// TIA Portal V16 program export: 2 tag tables, 1 data types, 0 data blocks, 8 code blocks (in call order from the OBs), 7 instance data blocks

VAR_GLOBAL   // PLC tag table "Default tag table"
END_VAR

VAR_GLOBAL   // PLC tag table "Outputs"
   qIO_xSupplyConveyor1 AT %Q0.0 : Bool;
   qIO_xSupplyConveyor2 AT %Q0.1 : Bool;
   qIO_xS1Conveyor1 AT %Q0.2 : Bool;
   qIO_xS1Conveyor2 AT %Q0.3 : Bool;
   qIO_xS1Conveyor3 AT %Q0.4 : Bool;
   qIO_xS1PositionerClamp AT %Q0.5 : Bool;
   qIO_xS1PositionerRaise AT %Q0.6 : Bool;
   qIO_xS2Conveyor1 AT %Q0.7 : Bool;
   qIO_xS2Conveyor2 AT %Q1.0 : Bool;
   qIO_xS2Conveyor3 AT %Q1.1 : Bool;
   qIO_xS2PositionerClamp AT %Q1.2 : Bool;
   qIO_xS2PositionerRaise AT %Q1.3 : Bool;
   qIO_xS3Conveyor1 AT %Q1.4 : Bool;
   qIO_xS3Conveyor2 AT %Q1.5 : Bool;
   qIO_xS3Conveyor3 AT %Q1.6 : Bool;
   qIO_xS3PositionerClamp AT %Q1.7 : Bool;
   qIO_xS3PositionerRaise AT %Q2.0 : Bool;
   qIO_xS1ProcessLight AT %Q2.1 : Bool;
   qIO_iS1ProcessTimeLeft AT %QD10 : DInt;
   qIO_xS2ProcessLight AT %Q2.2 : Bool;
   qIO_iS2ProcessTimeLeft AT %QD14 : DInt;
   qIO_xS3ProcessLight AT %Q2.3 : Bool;
   qIO_iS3ProcessTimeLeft AT %QD18 : DInt;
   qIO_xSupplyGetMaterial AT %Q2.4 : Bool;
END_VAR

TYPE "UDT SupplyStation"
// stored: IsFailsafeCompliant false
   STRUCT
      Status : Struct
         xSpare : Bool;
      END_STRUCT;
      Command : Struct
         xSupplyDataRequest : Bool;
      END_STRUCT;
      Fault : Struct
         xSpare : Bool;
      END_STRUCT;
   END_STRUCT;
END_TYPE

ORGANIZATION_BLOCK "Main"   // OB1, LAD, ProgramCycle
TITLE = "Main Program Sweep (Cycle)"
{ S7_Optimized_Access := 'TRUE' }
VERSION : 0.1
// stored: AutoNumber true, IsIECCheckEnabled false, SetENOAutomatically false
   VAR_INPUT
      Initial_Call : Bool;   // Initial call of this OB
      Remanence : Bool;   // =True, if remanent data are available
   END_VAR
   VAR_TEMP   // added for the SCL form of the ladder/FBD networks
      _w1 : Bool;
   END_VAR
BEGIN

REGION Network 1
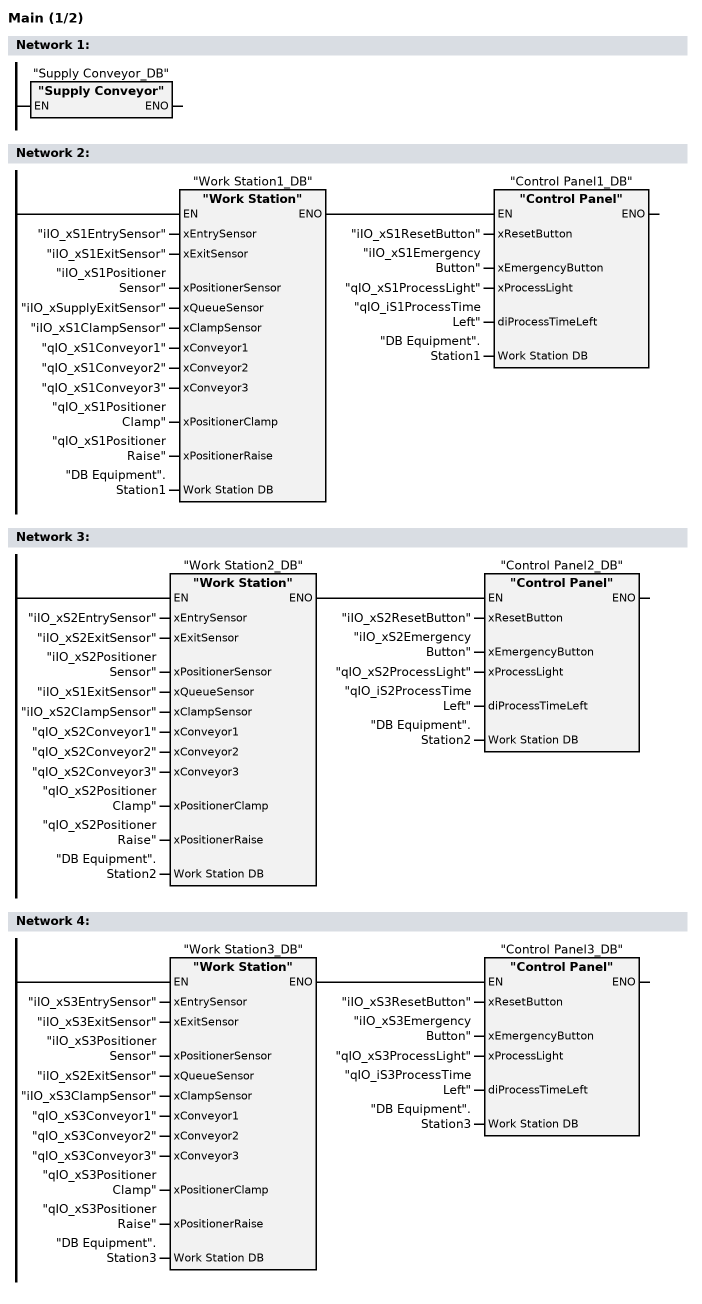
   RUNG wire#powerrail
      "Supply Conveyor_DB"()
   END_RUNG
   // the same network as SCL:
   "Supply Conveyor_DB"();   // "Supply Conveyor"
END_REGION

REGION Network 2
   RUNG wire#powerrail
      "Work Station1_DB"(xEntrySensor := "iIO_xS1EntrySensor", xExitSensor := "iIO_xS1ExitSensor", xPositionerSensor := "iIO_xS1PositionerSensor", xQueueSensor := "iIO_xSupplyExitSensor", xClampSensor := "iIO_xS1ClampSensor", xConveyor1 := "qIO_xS1Conveyor1", xConveyor2 := "qIO_xS1Conveyor2", xConveyor3 := "qIO_xS1Conveyor3", xPositionerClamp := "qIO_xS1PositionerClamp", xPositionerRaise := "qIO_xS1PositionerRaise", "Work Station DB" := "DB Equipment".Station1)
      "Control Panel1_DB"(xResetButton := "iIO_xS1ResetButton", xEmergencyButton := "iIO_xS1EmergencyButton", xProcessLight := "qIO_xS1ProcessLight", diProcessTimeLeft := "qIO_iS1ProcessTimeLeft", "Work Station DB" := "DB Equipment".Station1)
   END_RUNG
   // the same network as SCL:
   "Work Station1_DB"(xEntrySensor := "iIO_xS1EntrySensor",   // "Work Station"
                      xExitSensor := "iIO_xS1ExitSensor",
                      xPositionerSensor := "iIO_xS1PositionerSensor",
                      xQueueSensor := "iIO_xSupplyExitSensor",
                      xClampSensor := "iIO_xS1ClampSensor",
                      xConveyor1 := "qIO_xS1Conveyor1",
                      xConveyor2 := "qIO_xS1Conveyor2",
                      xConveyor3 := "qIO_xS1Conveyor3",
                      xPositionerClamp := "qIO_xS1PositionerClamp",
                      xPositionerRaise := "qIO_xS1PositionerRaise",
                      "Work Station DB" := "DB Equipment".Station1,
                      ENO => #_w1);
   IF #_w1 THEN
       "Control Panel1_DB"(xResetButton := "iIO_xS1ResetButton",   // "Control Panel"
                           xEmergencyButton := "iIO_xS1EmergencyButton",
                           xProcessLight := "qIO_xS1ProcessLight",
                           diProcessTimeLeft := "qIO_iS1ProcessTimeLeft",
                           "Work Station DB" := "DB Equipment".Station1);
   END_IF;
END_REGION

REGION Network 3
   RUNG wire#powerrail
      "Work Station2_DB"(xEntrySensor := "iIO_xS2EntrySensor", xExitSensor := "iIO_xS2ExitSensor", xPositionerSensor := "iIO_xS2PositionerSensor", xQueueSensor := "iIO_xS1ExitSensor", xClampSensor := "iIO_xS2ClampSensor", xConveyor1 := "qIO_xS2Conveyor1", xConveyor2 := "qIO_xS2Conveyor2", xConveyor3 := "qIO_xS2Conveyor3", xPositionerClamp := "qIO_xS2PositionerClamp", xPositionerRaise := "qIO_xS2PositionerRaise", "Work Station DB" := "DB Equipment".Station2)
      "Control Panel2_DB"(xResetButton := "iIO_xS2ResetButton", xEmergencyButton := "iIO_xS2EmergencyButton", xProcessLight := "qIO_xS2ProcessLight", diProcessTimeLeft := "qIO_iS2ProcessTimeLeft", "Work Station DB" := "DB Equipment".Station2)
   END_RUNG
   // the same network as SCL:
   "Work Station2_DB"(xEntrySensor := "iIO_xS2EntrySensor",   // "Work Station"
                      xExitSensor := "iIO_xS2ExitSensor",
                      xPositionerSensor := "iIO_xS2PositionerSensor",
                      xQueueSensor := "iIO_xS1ExitSensor",
                      xClampSensor := "iIO_xS2ClampSensor",
                      xConveyor1 := "qIO_xS2Conveyor1",
                      xConveyor2 := "qIO_xS2Conveyor2",
                      xConveyor3 := "qIO_xS2Conveyor3",
                      xPositionerClamp := "qIO_xS2PositionerClamp",
                      xPositionerRaise := "qIO_xS2PositionerRaise",
                      "Work Station DB" := "DB Equipment".Station2,
                      ENO => #_w1);
   IF #_w1 THEN
       "Control Panel2_DB"(xResetButton := "iIO_xS2ResetButton",   // "Control Panel"
                           xEmergencyButton := "iIO_xS2EmergencyButton",
                           xProcessLight := "qIO_xS2ProcessLight",
                           diProcessTimeLeft := "qIO_iS2ProcessTimeLeft",
                           "Work Station DB" := "DB Equipment".Station2);
   END_IF;
END_REGION

REGION Network 4
   RUNG wire#powerrail
      "Work Station3_DB"(xEntrySensor := "iIO_xS3EntrySensor", xExitSensor := "iIO_xS3ExitSensor", xPositionerSensor := "iIO_xS3PositionerSensor", xQueueSensor := "iIO_xS2ExitSensor", xClampSensor := "iIO_xS3ClampSensor", xConveyor1 := "qIO_xS3Conveyor1", xConveyor2 := "qIO_xS3Conveyor2", xConveyor3 := "qIO_xS3Conveyor3", xPositionerClamp := "qIO_xS3PositionerClamp", xPositionerRaise := "qIO_xS3PositionerRaise", "Work Station DB" := "DB Equipment".Station3)
      "Control Panel3_DB"(xResetButton := "iIO_xS3ResetButton", xEmergencyButton := "iIO_xS3EmergencyButton", xProcessLight := "qIO_xS3ProcessLight", diProcessTimeLeft := "qIO_iS3ProcessTimeLeft", "Work Station DB" := "DB Equipment".Station3)
   END_RUNG
   // the same network as SCL:
   "Work Station3_DB"(xEntrySensor := "iIO_xS3EntrySensor",   // "Work Station"
                      xExitSensor := "iIO_xS3ExitSensor",
                      xPositionerSensor := "iIO_xS3PositionerSensor",
                      xQueueSensor := "iIO_xS2ExitSensor",
                      xClampSensor := "iIO_xS3ClampSensor",
                      xConveyor1 := "qIO_xS3Conveyor1",
                      xConveyor2 := "qIO_xS3Conveyor2",
                      xConveyor3 := "qIO_xS3Conveyor3",
                      xPositionerClamp := "qIO_xS3PositionerClamp",
                      xPositionerRaise := "qIO_xS3PositionerRaise",
                      "Work Station DB" := "DB Equipment".Station3,
                      ENO => #_w1);
   IF #_w1 THEN
       "Control Panel3_DB"(xResetButton := "iIO_xS3ResetButton",   // "Control Panel"
                           xEmergencyButton := "iIO_xS3EmergencyButton",
                           xProcessLight := "qIO_xS3ProcessLight",
                           diProcessTimeLeft := "qIO_iS3ProcessTimeLeft",
                           "Work Station DB" := "DB Equipment".Station3);
   END_IF;
END_REGION

REGION Network 5
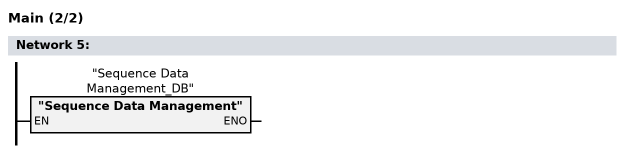
   RUNG wire#powerrail
      "Sequence Data Management_DB"()
   END_RUNG
   // the same network as SCL:
   "Sequence Data Management_DB"();   // "Sequence Data Management"
END_REGION
END_ORGANIZATION_BLOCK

FUNCTION_BLOCK "Work Station"   // FB1, LAD
{ S7_Optimized_Access := 'TRUE' }
VERSION : 0.1
// stored: AutoNumber true, IsIECCheckEnabled false, IsRetainMemResEnabled false, MemoryReserve 100, SetENOAutomatically false, UDAEnableTagReadback false
   VAR_INPUT
      xEntrySensor { ExternalAccessible := 'False'; ExternalVisible := 'False'; ExternalWritable := 'False'} : Bool;
      xExitSensor { ExternalAccessible := 'False'; ExternalVisible := 'False'; ExternalWritable := 'False'} : Bool;
      xPositionerSensor { ExternalAccessible := 'False'; ExternalVisible := 'False'; ExternalWritable := 'False'} : Bool;
      xQueueSensor { ExternalAccessible := 'False'; ExternalVisible := 'False'; ExternalWritable := 'False'} : Bool;
      xClampSensor { ExternalAccessible := 'False'; ExternalVisible := 'False'; ExternalWritable := 'False'} : Bool;
   END_VAR
   VAR_IN_OUT
      xConveyor1 { ExternalAccessible := 'False'; ExternalVisible := 'False'; ExternalWritable := 'False'} : Bool;
      xConveyor2 { ExternalAccessible := 'False'; ExternalVisible := 'False'; ExternalWritable := 'False'} : Bool;
      xConveyor3 { ExternalAccessible := 'False'; ExternalVisible := 'False'; ExternalWritable := 'False'} : Bool;
      xPositionerClamp : Bool;
      xPositionerRaise : Bool;
      "Work Station DB" : "UDT WorkStation";
   END_VAR
   VAR
      StationConveyorControl_Instance { S7_SetPoint := 'True'} : "StationConveyorControl";
      StationProcessControl_Instance { S7_SetPoint := 'True'} : "StationProcessControl";
   END_VAR
BEGIN

REGION Network 2
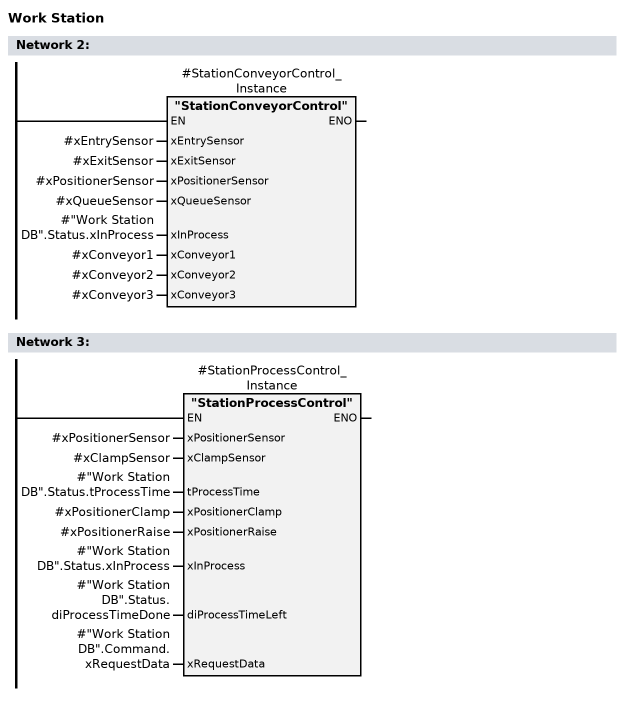
   RUNG wire#powerrail
      #StationConveyorControl_Instance(xEntrySensor := #xEntrySensor, xExitSensor := #xExitSensor, xPositionerSensor := #xPositionerSensor, xQueueSensor := #xQueueSensor, xInProcess := #"Work Station DB".Status.xInProcess, xConveyor1 := #xConveyor1, xConveyor2 := #xConveyor2, xConveyor3 := #xConveyor3)
   END_RUNG
   // the same network as SCL:
   #StationConveyorControl_Instance(xEntrySensor := #xEntrySensor,   // "StationConveyorControl"
                           xExitSensor := #xExitSensor,
                           xPositionerSensor := #xPositionerSensor,
                           xQueueSensor := #xQueueSensor,
                           xInProcess := #"Work Station DB".Status.xInProcess,
                           xConveyor1 := #xConveyor1,
                           xConveyor2 := #xConveyor2,
                           xConveyor3 := #xConveyor3);
END_REGION

REGION Network 3
   RUNG wire#powerrail
      #StationProcessControl_Instance(xPositionerSensor := #xPositionerSensor, xClampSensor := #xClampSensor, tProcessTime := #"Work Station DB".Status.tProcessTime, xPositionerClamp := #xPositionerClamp, xPositionerRaise := #xPositionerRaise, xInProcess := #"Work Station DB".Status.xInProcess, diProcessTimeLeft := #"Work Station DB".Status.diProcessTimeDone, xRequestData := #"Work Station DB".Command.xRequestData)
   END_RUNG
   // the same network as SCL:
   #StationProcessControl_Instance(xPositionerSensor := #xPositionerSensor,   // "StationProcessControl"
                           xClampSensor := #xClampSensor,
                           tProcessTime := #"Work Station DB".Status.tProcessTime,
                           xPositionerClamp := #xPositionerClamp,
                           xPositionerRaise := #xPositionerRaise,
                           xInProcess := #"Work Station DB".Status.xInProcess,
                           diProcessTimeLeft := #"Work Station DB".Status.diProcessTimeDone,
                           xRequestData := #"Work Station DB".Command.xRequestData);
END_REGION
END_FUNCTION_BLOCK

FUNCTION_BLOCK "StationProcessControl"   // FB4, LAD
{ S7_Optimized_Access := 'TRUE' }
VERSION : 0.1
// stored: AutoNumber true, IsIECCheckEnabled false, IsRetainMemResEnabled false, MemoryReserve 100, SetENOAutomatically false, UDAEnableTagReadback false
   VAR_INPUT
      xPositionerSensor { ExternalAccessible := 'False'; ExternalVisible := 'False'; ExternalWritable := 'False'} : Bool;
      xClampSensor { ExternalAccessible := 'False'; ExternalVisible := 'False'; ExternalWritable := 'False'} : Bool;
      tProcessTime { ExternalAccessible := 'False'; ExternalVisible := 'False'; ExternalWritable := 'False'} : Time;
   END_VAR
   VAR_IN_OUT
      xPositionerClamp : Bool;
      xPositionerRaise : Bool;
      xInProcess : Bool;
      diProcessTimeLeft : DInt;
      xRequestData : Bool;
   END_VAR
   VAR
      xProcessDone : Bool := false;
      xEdgeMemory1 : Bool;
      xEdgeMemory2 : Bool := false;
      IEC_Timer_0_Instance { S7_SetPoint := 'True'} : TON_TIME;
   END_VAR
   VAR_TEMP   // added for the SCL form of the ladder/FBD networks
      _w1 : Bool;
   END_VAR
BEGIN

REGION Network 1: Clamp positioner if material is detected, request for data
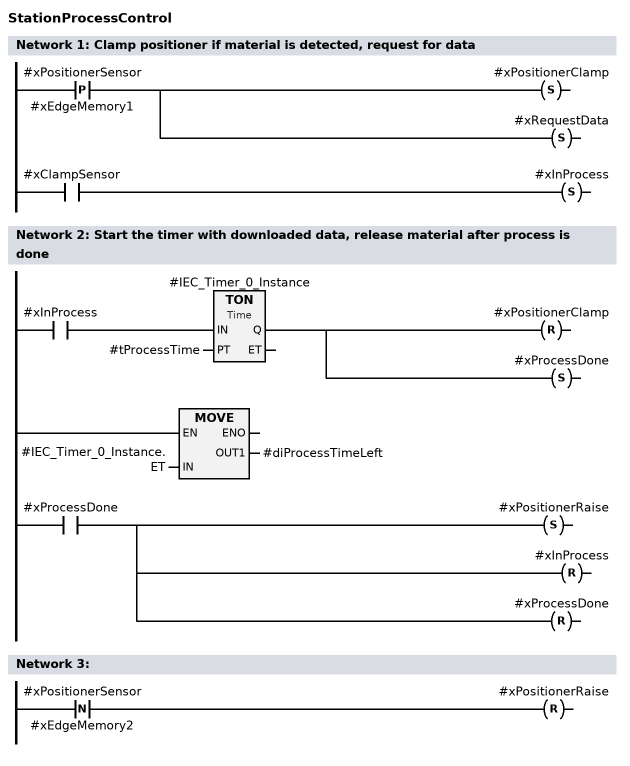
   RUNG wire#powerrail
      P_Contact(operand := #xPositionerSensor, bit := #xEdgeMemory1)
      wire#w1
      S_Coil( #xPositionerClamp )
   END_RUNG
   RUNG wire#w1
      S_Coil( #xRequestData )
   END_RUNG
   RUNG wire#powerrail
      Contact( #xClampSensor )
      S_Coil( #xInProcess )
   END_RUNG
   // the same network as SCL:
   #_w1 := #xPositionerSensor AND NOT #xEdgeMemory1;   // rising edge of #xPositionerSensor
   #xEdgeMemory1 := #xPositionerSensor;
   IF #_w1 THEN
       #xPositionerClamp := TRUE;
       #xRequestData := TRUE;
   END_IF;
   IF #xClampSensor THEN #xInProcess := TRUE; END_IF;
END_REGION

REGION Network 2: Start the timer with downloaded data, release material after process is done
   RUNG wire#powerrail
      Contact( #xInProcess )
      { S7_Templates := "time_type := Time" } #IEC_Timer_0_Instance.TON(pt := #tProcessTime, et =>)
      wire#w1
      R_Coil( #xPositionerClamp )
   END_RUNG
   RUNG wire#w1
      S_Coil( #xProcessDone )
   END_RUNG
   RUNG wire#powerrail
      Move(in := #IEC_Timer_0_Instance.ET, out1 => #diProcessTimeLeft)
   END_RUNG
   RUNG wire#powerrail
      Contact( #xProcessDone )
      wire#w2
      S_Coil( #xPositionerRaise )
   END_RUNG
   RUNG wire#w2
      R_Coil( #xInProcess )
   END_RUNG
   RUNG wire#w2
      R_Coil( #xProcessDone )
   END_RUNG
   // the same network as SCL:
   #IEC_Timer_0_Instance(IN := #xInProcess, PT := #tProcessTime);   // TON
   IF #IEC_Timer_0_Instance.Q THEN
       #xPositionerClamp := FALSE;
       #xProcessDone := TRUE;
   END_IF;
   #diProcessTimeLeft := #IEC_Timer_0_Instance.ET;
   IF #xProcessDone THEN
       #xPositionerRaise := TRUE;
       #xInProcess := FALSE;
       #xProcessDone := FALSE;
   END_IF;
END_REGION

REGION Network 3
   RUNG wire#powerrail
      N_Contact(operand := #xPositionerSensor, bit := #xEdgeMemory2)
      R_Coil( #xPositionerRaise )
   END_RUNG
   // the same network as SCL:
   #_w1 := NOT #xPositionerSensor AND #xEdgeMemory2;   // falling edge of #xPositionerSensor
   #xEdgeMemory2 := #xPositionerSensor;
   IF #_w1 THEN #xPositionerRaise := FALSE; END_IF;
END_REGION
END_FUNCTION_BLOCK

FUNCTION_BLOCK "Control Panel"   // FB2, LAD
{ S7_Optimized_Access := 'TRUE' }
VERSION : 0.1
// stored: AutoNumber true, IsIECCheckEnabled false, IsRetainMemResEnabled false, MemoryReserve 100, SetENOAutomatically false, UDAEnableTagReadback false
   VAR_INPUT
      xResetButton : Bool;
      xEmergencyButton : Bool;
   END_VAR
   VAR_IN_OUT
      xProcessLight : Bool;
      diProcessTimeLeft : DInt;
      "Work Station DB" : "UDT WorkStation";
   END_VAR
   VAR
      diProcessTime : DInt;
   END_VAR
BEGIN

REGION Network 1
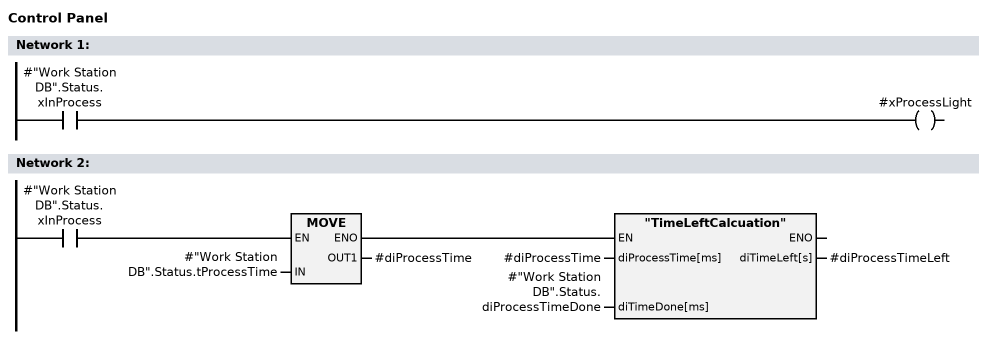
   RUNG wire#powerrail
      Contact( #"Work Station DB".Status.xInProcess )
      Coil( #xProcessLight )
   END_RUNG
   // the same network as SCL:
   #xProcessLight := #"Work Station DB".Status.xInProcess;
END_REGION

REGION Network 2
   RUNG wire#powerrail
      Contact( #"Work Station DB".Status.xInProcess )
      Move(in := #"Work Station DB".Status.tProcessTime, out1 => #diProcessTime)
      "TimeLeftCalcuation"("diProcessTime[ms]" := #diProcessTime, "diTimeDone[ms]" := #"Work Station DB".Status.diProcessTimeDone, "diTimeLeft[s]" => #diProcessTimeLeft)
   END_RUNG
   // the same network as SCL:
   IF #"Work Station DB".Status.xInProcess THEN
       #diProcessTime := #"Work Station DB".Status.tProcessTime;
       "TimeLeftCalcuation"("diProcessTime[ms]" := #diProcessTime,
                            "diTimeDone[ms]" := #"Work Station DB".Status.diProcessTimeDone,
                            "diTimeLeft[s]" => #diProcessTimeLeft);
   END_IF;
END_REGION
END_FUNCTION_BLOCK

FUNCTION "TimeLeftCalcuation" : Void
{ S7_Optimized_Access := 'TRUE' }
VERSION : 0.1
   VAR_INPUT 
      "diProcessTime[ms]" : DInt;
      "diTimeDone[ms]" : DInt;
   END_VAR

   VAR_OUTPUT 
      "diTimeLeft[s]" : DInt;
   END_VAR


BEGIN
	#"diTimeLeft[s]" := (#"diProcessTime[ms]" - #"diTimeDone[ms]") / 1000;
	
END_FUNCTION

FUNCTION_BLOCK "Sequence Data Management"   // FB3, LAD
{ S7_Optimized_Access := 'TRUE' }
VERSION : 0.1
// stored: AutoNumber true, IsIECCheckEnabled false, IsRetainMemResEnabled false, MemoryReserve 100, SetENOAutomatically false, UDAEnableTagReadback false
   VAR
      WorkStationList1 : Array[0..9] of DInt;
      WorkStationList2 : Array[0..9] of DInt;
      WorkStationList3 : Array[0..9] of DInt;
   END_VAR
   // WorkStationList1[0..9] := -1;
   // WorkStationList2[0..9] := -1;
   // WorkStationList3[0..9] := -1;
   VAR_TEMP   // added for the SCL form of the ladder/FBD networks
      _w1 : Bool;
      _w2 : Bool;
   END_VAR
BEGIN

REGION Network 1
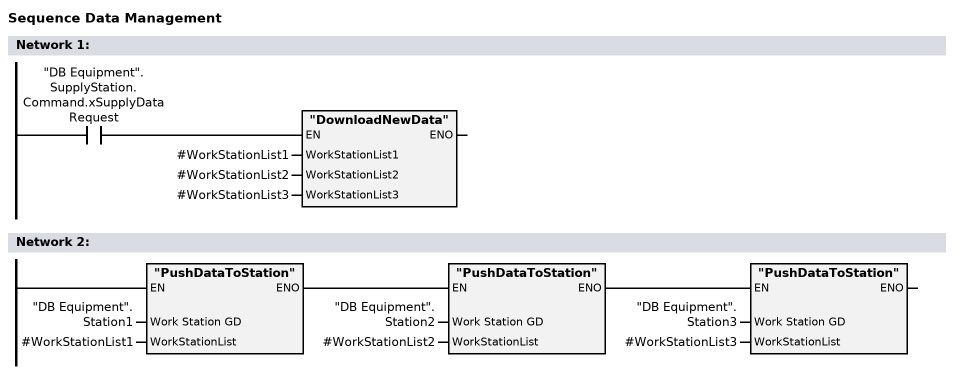
   RUNG wire#powerrail
      Contact( "DB Equipment".SupplyStation.Command.xSupplyDataRequest )
      "DownloadNewData"(WorkStationList1 := #WorkStationList1, WorkStationList2 := #WorkStationList2, WorkStationList3 := #WorkStationList3)
   END_RUNG
   // the same network as SCL:
   IF "DB Equipment".SupplyStation.Command.xSupplyDataRequest THEN
       "DownloadNewData"(WorkStationList1 := #WorkStationList1,
                         WorkStationList2 := #WorkStationList2,
                         WorkStationList3 := #WorkStationList3);
   END_IF;
END_REGION

REGION Network 2
   RUNG wire#powerrail
      "PushDataToStation"("Work Station GD" := "DB Equipment".Station1, WorkStationList := #WorkStationList1)
      "PushDataToStation"("Work Station GD" := "DB Equipment".Station2, WorkStationList := #WorkStationList2)
      "PushDataToStation"("Work Station GD" := "DB Equipment".Station3, WorkStationList := #WorkStationList3)
   END_RUNG
   // the same network as SCL:
   "PushDataToStation"("Work Station GD" := "DB Equipment".Station1,
                       WorkStationList := #WorkStationList1,
                       ENO => #_w1);
   "PushDataToStation"(EN := #_w1,
                       "Work Station GD" := "DB Equipment".Station2,
                       WorkStationList := #WorkStationList2,
                       ENO => #_w2);
   IF #_w2 THEN
       "PushDataToStation"("Work Station GD" := "DB Equipment".Station3, WorkStationList := #WorkStationList3);
   END_IF;
END_REGION
END_FUNCTION_BLOCK

FUNCTION "DownloadNewData" : Void
{ S7_Optimized_Access := 'TRUE' }
VERSION : 0.1
   VAR_IN_OUT 
      WorkStationList1 : Array[0..9] of DInt;
      WorkStationList2 : Array[0..9] of DInt;
      WorkStationList3 : Array[0..9] of DInt;
   END_VAR

   VAR_TEMP 
      iCounter1 : Int;
   END_VAR


BEGIN
	"DB Services".DataManager.Status.xTiaReady := true;
	
	IF "DB Services".DataManager.Status.xCReady THEN
	    //Push Data to arrays//
	    FOR #iCounter1 := 0 TO 9 DO
	        IF #WorkStationList1[#iCounter1] = -1 THEN
	            #WorkStationList1[#iCounter1] := "DB Services".DataManager.Status.DownloadedData[0];
	            EXIT;
	            ;
	        END_IF;
	        ;
	    END_FOR;
	    
	    FOR #iCounter1 := 0 TO 9 DO
	        IF #WorkStationList2[#iCounter1] = -1 THEN
	            #WorkStationList2[#iCounter1] := "DB Services".DataManager.Status.DownloadedData[1];
	            EXIT;
	            ;
	        END_IF;
	        ;
	    END_FOR;
	    
	    FOR #iCounter1 := 0 TO 9 DO
	        IF #WorkStationList3[#iCounter1] = -1 THEN
	            #WorkStationList3[#iCounter1] := "DB Services".DataManager.Status.DownloadedData[2];
	            EXIT;
	            ;
	        END_IF;
	        ;
	    END_FOR;
	    
	    "DB Services".DataManager.Status.xTiaReady := false;
	    "DB Services".DataManager.Status.xDataTransfered := true;
	    "DB Equipment".SupplyStation.Command.xSupplyDataRequest := false;
	END_IF;
	
	
	
	
END_FUNCTION

FUNCTION "PushDataToStation" : Void
{ S7_Optimized_Access := 'TRUE' }
VERSION : 0.1
   VAR_IN_OUT 
      "Work Station GD" : "UDT WorkStation";
      WorkStationList : Array[0..9] of DInt;
   END_VAR

   VAR_TEMP 
      iArrayLength : Int;
      iTemp : Int;
      iCounter : Int;
   END_VAR


BEGIN
	IF #"Work Station GD".Command.xRequestData THEN
	    #"Work Station GD".Status.tProcessTime := DINT_TO_TIME(#WorkStationList[0] * 1000);
	    #"Work Station GD".Command.xRequestData := false;
	    
	    FOR #iCounter := 0 TO 8  DO
	        #WorkStationList[#iCounter] := #WorkStationList[#iCounter + 1];
	        ;
	    END_FOR;
	    
	    ;
	END_IF;
	
END_FUNCTION

DATA_BLOCK "Control Panel1_DB"   // DB2
VERSION : 0.1
// stored: AutoNumber true, DBAccessibleFromOPCUA true, InstanceOfName Control Panel, InstanceOfType FB
"Control Panel"
BEGIN
END_DATA_BLOCK

DATA_BLOCK "Control Panel2_DB"   // DB8
VERSION : 0.1
// stored: AutoNumber true, DBAccessibleFromOPCUA true, InstanceOfName Control Panel, InstanceOfType FB
"Control Panel"
BEGIN
END_DATA_BLOCK

DATA_BLOCK "Control Panel3_DB"   // DB9
VERSION : 0.1
// stored: AutoNumber true, DBAccessibleFromOPCUA true, InstanceOfName Control Panel, InstanceOfType FB
"Control Panel"
BEGIN
END_DATA_BLOCK

DATA_BLOCK "Supply Conveyor_DB"   // DB6
VERSION : 0.1
// stored: AutoNumber true, DBAccessibleFromOPCUA true, InstanceOfName Supply Conveyor, InstanceOfType FB
"Supply Conveyor"
   // VAR
   //    xMaterialOnConveyor : Bool;
   //    xEdgeMemory1 { ExternalAccessible := 'False'; ExternalVisible := 'False'; ExternalWritable := 'False'} : Bool;
   //    xEdgeMemory2 { ExternalAccessible := 'False'; ExternalVisible := 'False'; ExternalWritable := 'False'} : Bool;
   //    xEdgeMemory3 { ExternalAccessible := 'False'; ExternalVisible := 'False'; ExternalWritable := 'False'} : Bool;
   // END_VAR
BEGIN
END_DATA_BLOCK

DATA_BLOCK "Work Station1_DB"   // DB1
VERSION : 0.1
// stored: AutoNumber true, DBAccessibleFromOPCUA true, InstanceOfName Work Station, InstanceOfType FB
"Work Station"
BEGIN
END_DATA_BLOCK

DATA_BLOCK "Work Station2_DB"   // DB7
VERSION : 0.1
// stored: AutoNumber true, DBAccessibleFromOPCUA true, InstanceOfName Work Station, InstanceOfType FB
"Work Station"
BEGIN
END_DATA_BLOCK

DATA_BLOCK "Work Station3_DB"   // DB3
VERSION : 0.1
// stored: AutoNumber true, DBAccessibleFromOPCUA true, InstanceOfName Work Station, InstanceOfType FB
"Work Station"
BEGIN
END_DATA_BLOCK
